FUNCTION_BLOCK STR_Param
VAR_INPUT PERSISTENT
	val			: Strings.Str;
END_VAR

END_FUNCTION_BLOCK

(* stored: Version 1.1.0.1
   POU STR_Param: Id {1639af2c-84d4-403a-a531-06372bf02e4e}, SpecialFunc None *)
